GLOBALCONSTANTS ISO_CAN_NODE (* Global constants *)
  (* Standard: 61499-1 *)
  (* Version 1.0, 2025-10-05, franz *)
  PACKAGE isobus::pgn;
  VAR_GLOBAL CONSTANT
    NODE1 : USINT := 0; (* CAN 1 *)
    NODE2 : USINT := 1; (* CAN 2 *)
    NODE3 : USINT := 2; (* CAN 3 *)
    NODE4 : USINT := 3; (* CAN 4 *)
    INVALID : USINT := USINT#16#FF; (* CAN Invalid *)
  END_VAR
END_GLOBALCONSTANTS
